TYPE "Positioning_DOL_Machine_DataOut"
VERSION : 0.1
// Block: Positioning_DOL_Machine_DataOut
   STRUCT
      Fan_M_Contactor : Bool;
   END_STRUCT;

END_TYPE
